# EPICS substitutions: SKFMB350/SKFMB350-IOC-01App/Db/chopper.substitutions
file chopper.template {

pattern {PORT, P, CRATE}
{"\$(PORT)", "\$(P)", "1"}
{"\$(PORT)", "\$(P)", "2"}
}
